{attribute 'GeneratedUsingTerminal: EJ7211-0011-0026'}
{attribute addProperty BoxType "EJ7211-0011-0026"}
{attribute addProperty Id "Position_actual_valueAT %I*UDINT4"}
{attribute addProperty CRC "131878004"}
{attribute addProperty Size "4"}
TYPE DS402_Position_actual_value_07DC4C74 :
STRUCT
	{attribute addProperty Name "Position_actual_value"}
	Position_actual_value AT %I* : UDINT;
END_STRUCT
END_TYPE

(* stored: Version 1.2.0.0, ProductVersion 3.1.4024.9
   DUT DS402_Position_actual_value_07DC4C74: Id {a15f2d4f-fca1-4f42-9833-918474a4c88c} *)
